{attribute 'qualified_only'}
{attribute 'strict'}
TYPE OvenDoor :
(
	open := 0,
	close 
);
END_TYPE

(* stored: Version 1.1.0.1, ProductVersion 3.1.4022.12
   DUT OvenDoor: Id {10d9a00e-d63c-49e6-9773-a1fde86c534a} *)
